// TIA Portal V19 export
FUNCTION_BLOCK "F_Zone11_FB"   // FB178, F_LAD
TITLE = SAFETY ZONE 11 - AREA 02 (PROFILATRICE)
// -
// stored: Access Published
   VAR
      D10 : "Door_FB";
      D11 : "Door_FB";
      D12 : "Door_FB";
      FNS : "ForceNormalStop";
      F_Contactor_CambioFormato_Profilatrice { ExternalAccessible := 'False'; ExternalVisible := 'False'; ExternalWritable := 'False'} : "FDevice_Contactor_FB";
      F_Sinamics_Cassetta1_OP { ExternalAccessible := 'False'; ExternalVisible := 'False'; ExternalWritable := 'False'} : "FDevice_Sinamics_FB";
      F_Sinamics_Cassetta1_MOT { ExternalAccessible := 'False'; ExternalVisible := 'False'; ExternalWritable := 'False'} : "FDevice_Sinamics_FB";
      F_Sinamics_Cassetta2_OP { ExternalAccessible := 'False'; ExternalVisible := 'False'; ExternalWritable := 'False'} : "FDevice_Sinamics_FB";
      F_Sinamics_Cassetta2_MOT { ExternalAccessible := 'False'; ExternalVisible := 'False'; ExternalWritable := 'False'} : "FDevice_Sinamics_FB";
      F_Sinamics_Cassetta3_OP { ExternalAccessible := 'False'; ExternalVisible := 'False'; ExternalWritable := 'False'} : "FDevice_Sinamics_FB";
      F_Sinamics_Cassetta3_MOT { ExternalAccessible := 'False'; ExternalVisible := 'False'; ExternalWritable := 'False'} : "FDevice_Sinamics_FB";
   END_VAR
   VAR_TEMP
      DoorNormalStop : Bool;
      DoorSafeStop : Bool;
      Door_Ok : Bool;
   END_VAR
   VAR CONSTANT
      CASSETTE_S120_STOPPING_TIME : Time := T#1S;
   END_VAR
BEGIN

REGION Network 1: < < < < < < < < < < DOOR > > > > > > > > > >
END_REGION

REGION Network 2: Zone Entry enable
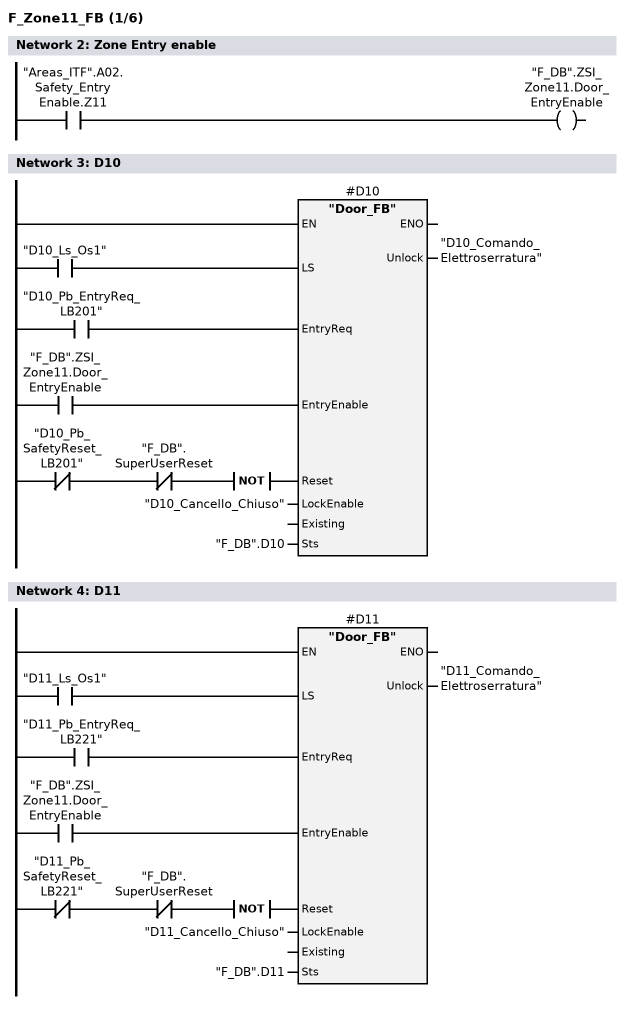
   RUNG wire#powerrail
      Contact( "Areas_ITF".A02.Safety_EntryEnable.Z11 )
      Coil( "F_DB".ZSI_Zone11.Door_EntryEnable )
   END_RUNG
   // the same network as SCL:
   "F_DB".ZSI_Zone11.Door_EntryEnable := "Areas_ITF".A02.Safety_EntryEnable.Z11;
END_REGION

REGION Network 3: D10
   RUNG wire#powerrail
      #D10(LS := wire#w1, EntryReq := wire#w2, EntryEnable := wire#w3, Reset := wire#w4, LockEnable := "D10_Cancello_Chiuso", Existing :=, Sts := "F_DB".D10, Unlock => "D10_Comando_Elettroserratura")
   END_RUNG
   RUNG wire#powerrail
      Contact( "D10_Ls_Os1" )
   END_RUNG wire#w1
   RUNG wire#powerrail
      Contact( "D10_Pb_EntryReq_LB201" )
   END_RUNG wire#w2
   RUNG wire#powerrail
      Contact( "F_DB".ZSI_Zone11.Door_EntryEnable )
   END_RUNG wire#w3
   RUNG wire#powerrail
      I_Contact( "D10_Pb_SafetyReset_LB201" )
      I_Contact( "F_DB".SuperUserReset )
      Not()
   END_RUNG wire#w4
   // the same network as SCL:
   #D10(LS := "D10_Ls_Os1",   // "Door_FB"
        EntryReq := "D10_Pb_EntryReq_LB201",
        EntryEnable := "F_DB".ZSI_Zone11.Door_EntryEnable,
        Reset := NOT (NOT "D10_Pb_SafetyReset_LB201" AND NOT "F_DB".SuperUserReset),
        LockEnable := "D10_Cancello_Chiuso",
        Sts := "F_DB".D10,
        Unlock => "D10_Comando_Elettroserratura");
END_REGION

REGION Network 4: D11
   RUNG wire#powerrail
      #D11(LS := wire#w1, EntryReq := wire#w2, EntryEnable := wire#w3, Reset := wire#w4, LockEnable := "D11_Cancello_Chiuso", Existing :=, Sts := "F_DB".D11, Unlock => "D11_Comando_Elettroserratura")
   END_RUNG
   RUNG wire#powerrail
      Contact( "D11_Ls_Os1" )
   END_RUNG wire#w1
   RUNG wire#powerrail
      Contact( "D11_Pb_EntryReq_LB221" )
   END_RUNG wire#w2
   RUNG wire#powerrail
      Contact( "F_DB".ZSI_Zone11.Door_EntryEnable )
   END_RUNG wire#w3
   RUNG wire#powerrail
      I_Contact( "D11_Pb_SafetyReset_LB221" )
      I_Contact( "F_DB".SuperUserReset )
      Not()
   END_RUNG wire#w4
   // the same network as SCL:
   #D11(LS := "D11_Ls_Os1",   // "Door_FB"
        EntryReq := "D11_Pb_EntryReq_LB221",
        EntryEnable := "F_DB".ZSI_Zone11.Door_EntryEnable,
        Reset := NOT (NOT "D11_Pb_SafetyReset_LB221" AND NOT "F_DB".SuperUserReset),
        LockEnable := "D11_Cancello_Chiuso",
        Sts := "F_DB".D11,
        Unlock => "D11_Comando_Elettroserratura");
END_REGION

REGION Network 5: D12
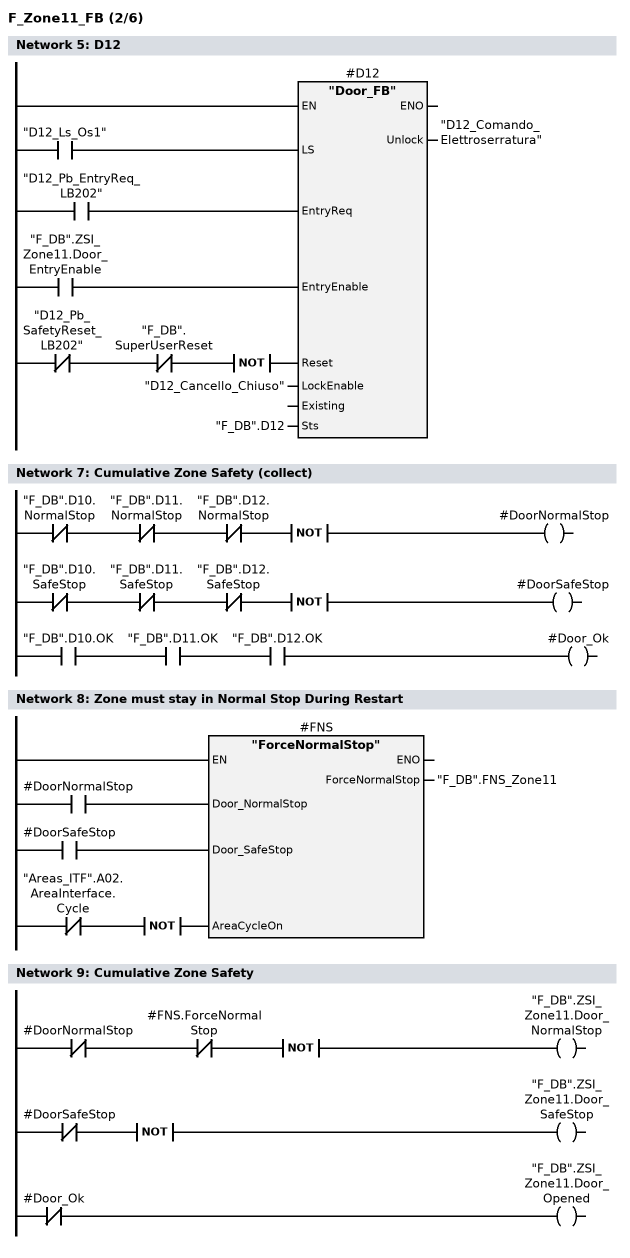
   RUNG wire#powerrail
      #D12(LS := wire#w1, EntryReq := wire#w2, EntryEnable := wire#w3, Reset := wire#w4, LockEnable := "D12_Cancello_Chiuso", Existing :=, Sts := "F_DB".D12, Unlock => "D12_Comando_Elettroserratura")
   END_RUNG
   RUNG wire#powerrail
      Contact( "D12_Ls_Os1" )
   END_RUNG wire#w1
   RUNG wire#powerrail
      Contact( "D12_Pb_EntryReq_LB202" )
   END_RUNG wire#w2
   RUNG wire#powerrail
      Contact( "F_DB".ZSI_Zone11.Door_EntryEnable )
   END_RUNG wire#w3
   RUNG wire#powerrail
      I_Contact( "D12_Pb_SafetyReset_LB202" )
      I_Contact( "F_DB".SuperUserReset )
      Not()
   END_RUNG wire#w4
   // the same network as SCL:
   #D12(LS := "D12_Ls_Os1",   // "Door_FB"
        EntryReq := "D12_Pb_EntryReq_LB202",
        EntryEnable := "F_DB".ZSI_Zone11.Door_EntryEnable,
        Reset := NOT (NOT "D12_Pb_SafetyReset_LB202" AND NOT "F_DB".SuperUserReset),
        LockEnable := "D12_Cancello_Chiuso",
        Sts := "F_DB".D12,
        Unlock => "D12_Comando_Elettroserratura");
END_REGION

REGION Network 6: < < < < < < < < < < ZONE SAFETY INTERFACE > > > > > > > > > >
END_REGION

REGION Network 7: Cumulative Zone Safety (collect)
   RUNG wire#powerrail
      I_Contact( "F_DB".D10.NormalStop )
      I_Contact( "F_DB".D11.NormalStop )
      I_Contact( "F_DB".D12.NormalStop )
      Not()
      Coil( #DoorNormalStop )
   END_RUNG
   RUNG wire#powerrail
      I_Contact( "F_DB".D10.SafeStop )
      I_Contact( "F_DB".D11.SafeStop )
      I_Contact( "F_DB".D12.SafeStop )
      Not()
      Coil( #DoorSafeStop )
   END_RUNG
   RUNG wire#powerrail
      Contact( "F_DB".D10.OK )
      Contact( "F_DB".D11.OK )
      Contact( "F_DB".D12.OK )
      Coil( #Door_Ok )
   END_RUNG
   // the same network as SCL:
   #DoorNormalStop := NOT (NOT "F_DB".D10.NormalStop AND NOT "F_DB".D11.NormalStop AND NOT "F_DB".D12.NormalStop);
   #DoorSafeStop := NOT (NOT "F_DB".D10.SafeStop AND NOT "F_DB".D11.SafeStop AND NOT "F_DB".D12.SafeStop);
   #Door_Ok := "F_DB".D10.OK AND "F_DB".D11.OK AND "F_DB".D12.OK;
END_REGION

REGION Network 8: Zone must stay in Normal Stop During Restart
   RUNG wire#powerrail
      #FNS(Door_NormalStop := wire#w1, Door_SafeStop := wire#w2, AreaCycleOn := wire#w3, ForceNormalStop => "F_DB".FNS_Zone11)
   END_RUNG
   RUNG wire#powerrail
      Contact( #DoorNormalStop )
   END_RUNG wire#w1
   RUNG wire#powerrail
      Contact( #DoorSafeStop )
   END_RUNG wire#w2
   RUNG wire#powerrail
      I_Contact( "Areas_ITF".A02.AreaInterface.Cycle )
      Not()
   END_RUNG wire#w3
   // the same network as SCL:
   #FNS(Door_NormalStop := #DoorNormalStop,   // "ForceNormalStop"
        Door_SafeStop := #DoorSafeStop,
        AreaCycleOn := NOT (NOT "Areas_ITF".A02.AreaInterface.Cycle),
        ForceNormalStop => "F_DB".FNS_Zone11);
END_REGION

REGION Network 9: Cumulative Zone Safety
   RUNG wire#powerrail
      I_Contact( #DoorNormalStop )
      I_Contact( #FNS.ForceNormalStop )
      Not()
      Coil( "F_DB".ZSI_Zone11.Door_NormalStop )
   END_RUNG
   RUNG wire#powerrail
      I_Contact( #DoorSafeStop )
      Not()
      Coil( "F_DB".ZSI_Zone11.Door_SafeStop )
   END_RUNG
   RUNG wire#powerrail
      I_Contact( #Door_Ok )
      Coil( "F_DB".ZSI_Zone11.Door_Opened )
   END_RUNG
   // the same network as SCL:
   "F_DB".ZSI_Zone11.Door_NormalStop := NOT (NOT #DoorNormalStop AND NOT #FNS.ForceNormalStop);
   "F_DB".ZSI_Zone11.Door_SafeStop := NOT (NOT #DoorSafeStop);
   "F_DB".ZSI_Zone11.Door_Opened := NOT #Door_Ok;
END_REGION

REGION Network 10: >
END_REGION

REGION Network 11: >
END_REGION

REGION Network 12: < < < < < < < < < < DEVICES SAFETY VALVES > > > > > > > > > >
END_REGION

REGION Network 13: >
END_REGION

REGION Network 14: >
END_REGION

REGION Network 15: < < < < < < < < < < DEVICES CONTACTORS > > > > > > > > > >
END_REGION

REGION Network 16: Contattore - Cambio formato Profilatrice
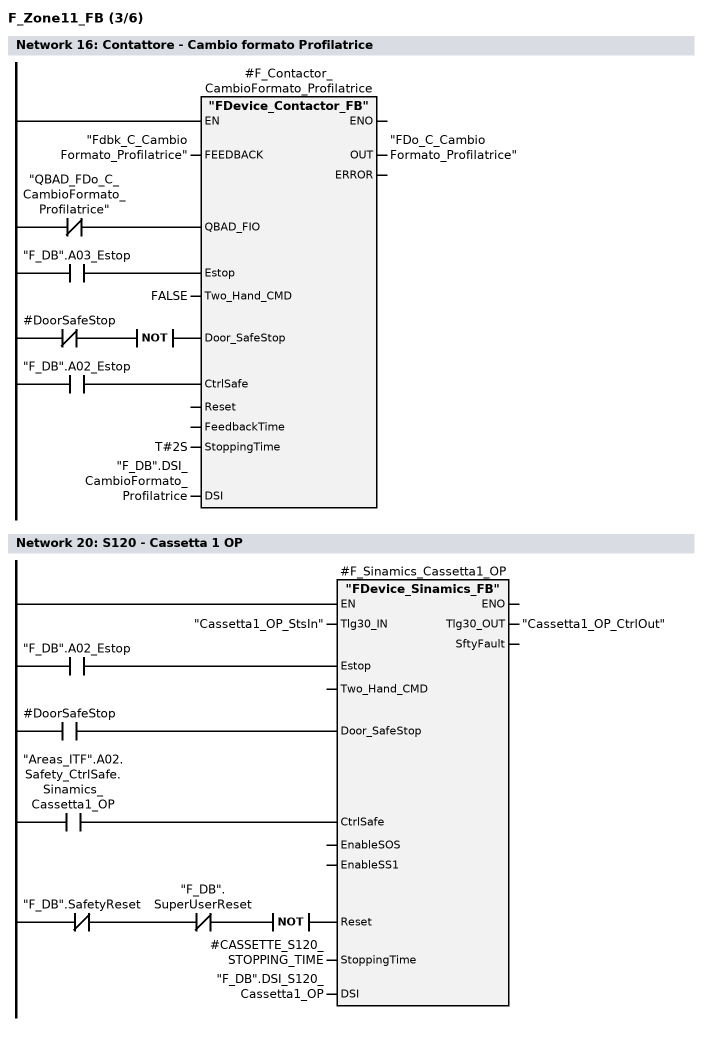
   RUNG wire#powerrail
      #F_Contactor_CambioFormato_Profilatrice(QBAD_FIO := wire#w1, Estop := wire#w2, Door_SafeStop := wire#w3, CtrlSafe := wire#w4, FEEDBACK := "Fdbk_C_CambioFormato_Profilatrice", Two_Hand_CMD := FALSE, Reset :=, FeedbackTime :=, StoppingTime := T#2S, DSI := "F_DB".DSI_CambioFormato_Profilatrice, OUT => "FDo_C_CambioFormato_Profilatrice", ERROR =>)
   END_RUNG
   RUNG wire#powerrail
      I_Contact( "QBAD_FDo_C_CambioFormato_Profilatrice" )
   END_RUNG wire#w1
   RUNG wire#powerrail
      Contact( "F_DB".A03_Estop )
   END_RUNG wire#w2
   RUNG wire#powerrail
      I_Contact( #DoorSafeStop )
      Not()
   END_RUNG wire#w3
   RUNG wire#powerrail
      Contact( "F_DB".A02_Estop )
   END_RUNG wire#w4
   // the same network as SCL:
   #F_Contactor_CambioFormato_Profilatrice(FEEDBACK := "Fdbk_C_CambioFormato_Profilatrice",   // "FDevice_Contactor_FB"
                           QBAD_FIO := NOT "QBAD_FDo_C_CambioFormato_Profilatrice",
                           Estop := "F_DB".A03_Estop,
                           Two_Hand_CMD := FALSE,
                           Door_SafeStop := NOT (NOT #DoorSafeStop),
                           CtrlSafe := "F_DB".A02_Estop,
                           StoppingTime := T#2S,
                           DSI := "F_DB".DSI_CambioFormato_Profilatrice,
                           OUT => "FDo_C_CambioFormato_Profilatrice");
END_REGION

REGION Network 17: >
END_REGION

REGION Network 18: >
END_REGION

REGION Network 19: < < < < < < < < < < DEVICES S120 > > > > > > > > > >
END_REGION

REGION Network 20: S120 - Cassetta 1 OP
   RUNG wire#powerrail
      #F_Sinamics_Cassetta1_OP(Estop := wire#w1, Door_SafeStop := wire#w2, CtrlSafe := wire#w3, Reset := wire#w4, Tlg30_IN := "Cassetta1_OP_StsIn", Two_Hand_CMD :=, EnableSOS :=, EnableSS1 :=, StoppingTime := #CASSETTE_S120_STOPPING_TIME, DSI := "F_DB".DSI_S120_Cassetta1_OP, Tlg30_OUT => "Cassetta1_OP_CtrlOut", SftyFault =>)
   END_RUNG
   RUNG wire#powerrail
      Contact( "F_DB".A02_Estop )
   END_RUNG wire#w1
   RUNG wire#powerrail
      Contact( #DoorSafeStop )
   END_RUNG wire#w2
   RUNG wire#powerrail
      Contact( "Areas_ITF".A02.Safety_CtrlSafe.Sinamics_Cassetta1_OP )
   END_RUNG wire#w3
   RUNG wire#powerrail
      I_Contact( "F_DB".SafetyReset )
      I_Contact( "F_DB".SuperUserReset )
      Not()
   END_RUNG wire#w4
   // the same network as SCL:
   #F_Sinamics_Cassetta1_OP(Tlg30_IN := "Cassetta1_OP_StsIn",   // "FDevice_Sinamics_FB"
                           Estop := "F_DB".A02_Estop,
                           Door_SafeStop := #DoorSafeStop,
                           CtrlSafe := "Areas_ITF".A02.Safety_CtrlSafe.Sinamics_Cassetta1_OP,
                           Reset := NOT (NOT "F_DB".SafetyReset AND NOT "F_DB".SuperUserReset),
                           StoppingTime := #CASSETTE_S120_STOPPING_TIME,
                           DSI := "F_DB".DSI_S120_Cassetta1_OP,
                           Tlg30_OUT => "Cassetta1_OP_CtrlOut");
END_REGION

REGION Network 21: S120 - Cassetta 1 MOT
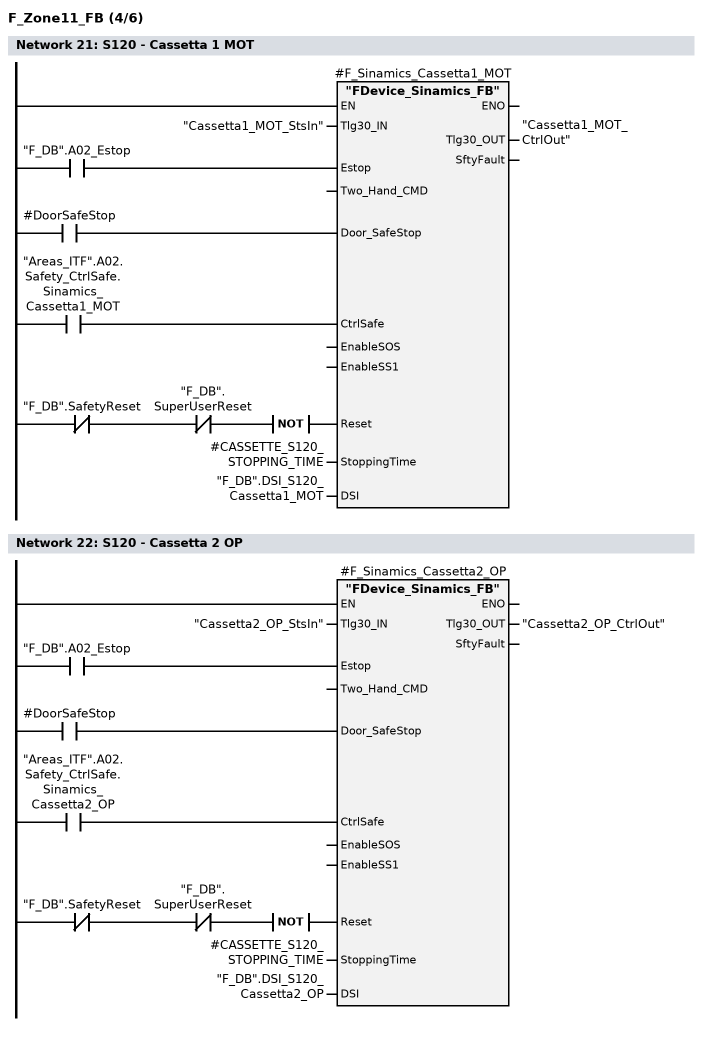
   RUNG wire#powerrail
      #F_Sinamics_Cassetta1_MOT(Estop := wire#w1, Door_SafeStop := wire#w2, CtrlSafe := wire#w3, Reset := wire#w4, Tlg30_IN := "Cassetta1_MOT_StsIn", Two_Hand_CMD :=, EnableSOS :=, EnableSS1 :=, StoppingTime := #CASSETTE_S120_STOPPING_TIME, DSI := "F_DB".DSI_S120_Cassetta1_MOT, Tlg30_OUT => "Cassetta1_MOT_CtrlOut", SftyFault =>)
   END_RUNG
   RUNG wire#powerrail
      Contact( "F_DB".A02_Estop )
   END_RUNG wire#w1
   RUNG wire#powerrail
      Contact( #DoorSafeStop )
   END_RUNG wire#w2
   RUNG wire#powerrail
      Contact( "Areas_ITF".A02.Safety_CtrlSafe.Sinamics_Cassetta1_MOT )
   END_RUNG wire#w3
   RUNG wire#powerrail
      I_Contact( "F_DB".SafetyReset )
      I_Contact( "F_DB".SuperUserReset )
      Not()
   END_RUNG wire#w4
   // the same network as SCL:
   #F_Sinamics_Cassetta1_MOT(Tlg30_IN := "Cassetta1_MOT_StsIn",   // "FDevice_Sinamics_FB"
                           Estop := "F_DB".A02_Estop,
                           Door_SafeStop := #DoorSafeStop,
                           CtrlSafe := "Areas_ITF".A02.Safety_CtrlSafe.Sinamics_Cassetta1_MOT,
                           Reset := NOT (NOT "F_DB".SafetyReset AND NOT "F_DB".SuperUserReset),
                           StoppingTime := #CASSETTE_S120_STOPPING_TIME,
                           DSI := "F_DB".DSI_S120_Cassetta1_MOT,
                           Tlg30_OUT => "Cassetta1_MOT_CtrlOut");
END_REGION

REGION Network 22: S120 - Cassetta 2 OP
   RUNG wire#powerrail
      #F_Sinamics_Cassetta2_OP(Estop := wire#w1, Door_SafeStop := wire#w2, CtrlSafe := wire#w3, Reset := wire#w4, Tlg30_IN := "Cassetta2_OP_StsIn", Two_Hand_CMD :=, EnableSOS :=, EnableSS1 :=, StoppingTime := #CASSETTE_S120_STOPPING_TIME, DSI := "F_DB".DSI_S120_Cassetta2_OP, Tlg30_OUT => "Cassetta2_OP_CtrlOut", SftyFault =>)
   END_RUNG
   RUNG wire#powerrail
      Contact( "F_DB".A02_Estop )
   END_RUNG wire#w1
   RUNG wire#powerrail
      Contact( #DoorSafeStop )
   END_RUNG wire#w2
   RUNG wire#powerrail
      Contact( "Areas_ITF".A02.Safety_CtrlSafe.Sinamics_Cassetta2_OP )
   END_RUNG wire#w3
   RUNG wire#powerrail
      I_Contact( "F_DB".SafetyReset )
      I_Contact( "F_DB".SuperUserReset )
      Not()
   END_RUNG wire#w4
   // the same network as SCL:
   #F_Sinamics_Cassetta2_OP(Tlg30_IN := "Cassetta2_OP_StsIn",   // "FDevice_Sinamics_FB"
                           Estop := "F_DB".A02_Estop,
                           Door_SafeStop := #DoorSafeStop,
                           CtrlSafe := "Areas_ITF".A02.Safety_CtrlSafe.Sinamics_Cassetta2_OP,
                           Reset := NOT (NOT "F_DB".SafetyReset AND NOT "F_DB".SuperUserReset),
                           StoppingTime := #CASSETTE_S120_STOPPING_TIME,
                           DSI := "F_DB".DSI_S120_Cassetta2_OP,
                           Tlg30_OUT => "Cassetta2_OP_CtrlOut");
END_REGION

REGION Network 23: S120 - Cassetta 2 MOT
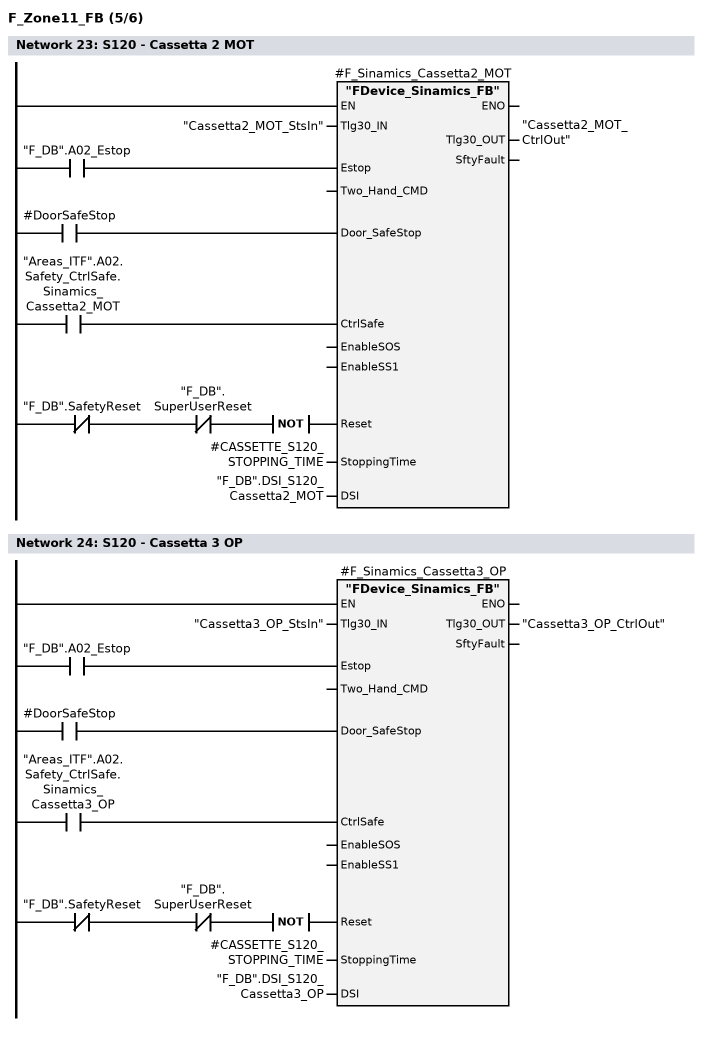
   RUNG wire#powerrail
      #F_Sinamics_Cassetta2_MOT(Estop := wire#w1, Door_SafeStop := wire#w2, CtrlSafe := wire#w3, Reset := wire#w4, Tlg30_IN := "Cassetta2_MOT_StsIn", Two_Hand_CMD :=, EnableSOS :=, EnableSS1 :=, StoppingTime := #CASSETTE_S120_STOPPING_TIME, DSI := "F_DB".DSI_S120_Cassetta2_MOT, Tlg30_OUT => "Cassetta2_MOT_CtrlOut", SftyFault =>)
   END_RUNG
   RUNG wire#powerrail
      Contact( "F_DB".A02_Estop )
   END_RUNG wire#w1
   RUNG wire#powerrail
      Contact( #DoorSafeStop )
   END_RUNG wire#w2
   RUNG wire#powerrail
      Contact( "Areas_ITF".A02.Safety_CtrlSafe.Sinamics_Cassetta2_MOT )
   END_RUNG wire#w3
   RUNG wire#powerrail
      I_Contact( "F_DB".SafetyReset )
      I_Contact( "F_DB".SuperUserReset )
      Not()
   END_RUNG wire#w4
   // the same network as SCL:
   #F_Sinamics_Cassetta2_MOT(Tlg30_IN := "Cassetta2_MOT_StsIn",   // "FDevice_Sinamics_FB"
                           Estop := "F_DB".A02_Estop,
                           Door_SafeStop := #DoorSafeStop,
                           CtrlSafe := "Areas_ITF".A02.Safety_CtrlSafe.Sinamics_Cassetta2_MOT,
                           Reset := NOT (NOT "F_DB".SafetyReset AND NOT "F_DB".SuperUserReset),
                           StoppingTime := #CASSETTE_S120_STOPPING_TIME,
                           DSI := "F_DB".DSI_S120_Cassetta2_MOT,
                           Tlg30_OUT => "Cassetta2_MOT_CtrlOut");
END_REGION

REGION Network 24: S120 - Cassetta 3 OP
   RUNG wire#powerrail
      #F_Sinamics_Cassetta3_OP(Estop := wire#w1, Door_SafeStop := wire#w2, CtrlSafe := wire#w3, Reset := wire#w4, Tlg30_IN := "Cassetta3_OP_StsIn", Two_Hand_CMD :=, EnableSOS :=, EnableSS1 :=, StoppingTime := #CASSETTE_S120_STOPPING_TIME, DSI := "F_DB".DSI_S120_Cassetta3_OP, Tlg30_OUT => "Cassetta3_OP_CtrlOut", SftyFault =>)
   END_RUNG
   RUNG wire#powerrail
      Contact( "F_DB".A02_Estop )
   END_RUNG wire#w1
   RUNG wire#powerrail
      Contact( #DoorSafeStop )
   END_RUNG wire#w2
   RUNG wire#powerrail
      Contact( "Areas_ITF".A02.Safety_CtrlSafe.Sinamics_Cassetta3_OP )
   END_RUNG wire#w3
   RUNG wire#powerrail
      I_Contact( "F_DB".SafetyReset )
      I_Contact( "F_DB".SuperUserReset )
      Not()
   END_RUNG wire#w4
   // the same network as SCL:
   #F_Sinamics_Cassetta3_OP(Tlg30_IN := "Cassetta3_OP_StsIn",   // "FDevice_Sinamics_FB"
                           Estop := "F_DB".A02_Estop,
                           Door_SafeStop := #DoorSafeStop,
                           CtrlSafe := "Areas_ITF".A02.Safety_CtrlSafe.Sinamics_Cassetta3_OP,
                           Reset := NOT (NOT "F_DB".SafetyReset AND NOT "F_DB".SuperUserReset),
                           StoppingTime := #CASSETTE_S120_STOPPING_TIME,
                           DSI := "F_DB".DSI_S120_Cassetta3_OP,
                           Tlg30_OUT => "Cassetta3_OP_CtrlOut");
END_REGION

REGION Network 25: S120 - Cassetta 3 MOT
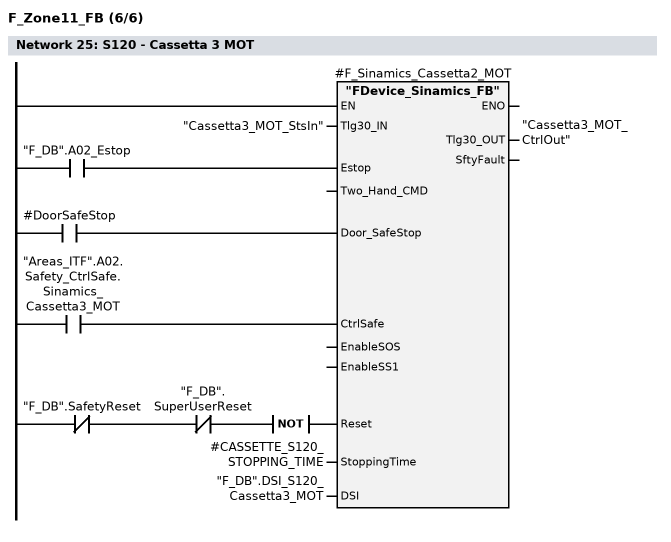
   RUNG wire#powerrail
      #F_Sinamics_Cassetta2_MOT(Estop := wire#w1, Door_SafeStop := wire#w2, CtrlSafe := wire#w3, Reset := wire#w4, Tlg30_IN := "Cassetta3_MOT_StsIn", Two_Hand_CMD :=, EnableSOS :=, EnableSS1 :=, StoppingTime := #CASSETTE_S120_STOPPING_TIME, DSI := "F_DB".DSI_S120_Cassetta3_MOT, Tlg30_OUT => "Cassetta3_MOT_CtrlOut", SftyFault =>)
   END_RUNG
   RUNG wire#powerrail
      Contact( "F_DB".A02_Estop )
   END_RUNG wire#w1
   RUNG wire#powerrail
      Contact( #DoorSafeStop )
   END_RUNG wire#w2
   RUNG wire#powerrail
      Contact( "Areas_ITF".A02.Safety_CtrlSafe.Sinamics_Cassetta3_MOT )
   END_RUNG wire#w3
   RUNG wire#powerrail
      I_Contact( "F_DB".SafetyReset )
      I_Contact( "F_DB".SuperUserReset )
      Not()
   END_RUNG wire#w4
   // the same network as SCL:
   #F_Sinamics_Cassetta2_MOT(Tlg30_IN := "Cassetta3_MOT_StsIn",   // "FDevice_Sinamics_FB"
                           Estop := "F_DB".A02_Estop,
                           Door_SafeStop := #DoorSafeStop,
                           CtrlSafe := "Areas_ITF".A02.Safety_CtrlSafe.Sinamics_Cassetta3_MOT,
                           Reset := NOT (NOT "F_DB".SafetyReset AND NOT "F_DB".SuperUserReset),
                           StoppingTime := #CASSETTE_S120_STOPPING_TIME,
                           DSI := "F_DB".DSI_S120_Cassetta3_MOT,
                           Tlg30_OUT => "Cassetta3_MOT_CtrlOut");
END_REGION

REGION Network 26: >
END_REGION

REGION Network 27: >
END_REGION
END_FUNCTION_BLOCK
